Omron CX-Programmer project NewProject (CX-Programmer 9.73)

# PLC NewPLC1: CJ1M CPU11

## Global symbols (name address type ; comment)
At_exit_forward 0.10 BOOL
At_exit_left 0.09 BOOL
At_exit_right 0.11 BOOL
At_forward_entry 0.07 BOOL
At_left_entry 0.06 BOOL
At_right_entry 0.08 BOOL
At_scale 0.04 BOOL
At_scale_entry 0.03 BOOL
At_scale_exit 0.05 BOOL
W200 CHANNEL  ; weight_help
Emergency 0.02 BOOL
Entry_conveyor W1.00 BOOL
Entry_conveyor_act 1.00 BOOL  ; Entry_conveyor
Forward_conveyor W1.03 BOOL
Forward_conveyor_act 1.03 BOOL
Forward_counter W301 INT
Forward_screen 2 CHANNEL
Left_conveyor W1.02 BOOL
Left_conveyor_act 1.02 BOOL
Left_counter W300 INT
Left_screen 1 CHANNEL
Load_scale W1.01 BOOL
Load_scale_act 1.01 BOOL
Mid W100 INT
Mid_flag W1.05 BOOL
On_forward_conveyor W304 INT
On_forward_conveyor_minus W1.08 BOOL
On_left_conveyor W303 INT
On_left_conveyor_minus W1.07 BOOL
On_load_scale W306 INT
On_load_scale_minus W1.06 BOOL
On_right_conveyor W305 INT
On_right_conveyor_minus W1.09 BOOL
Program_entry W0.01 BOOL
Right_conveyor W1.04 BOOL
Right_conveyor_act 1.04 BOOL
Right_counter W302 INT
Right_screen 3 CHANNEL
Start 0.00 BOOL  ; start
Stop 0.01 BOOL
Weight W0 INT  ; weight
Weight_screen 4 CHANNEL

## Program weight_sorter_program (cyclic task 1)
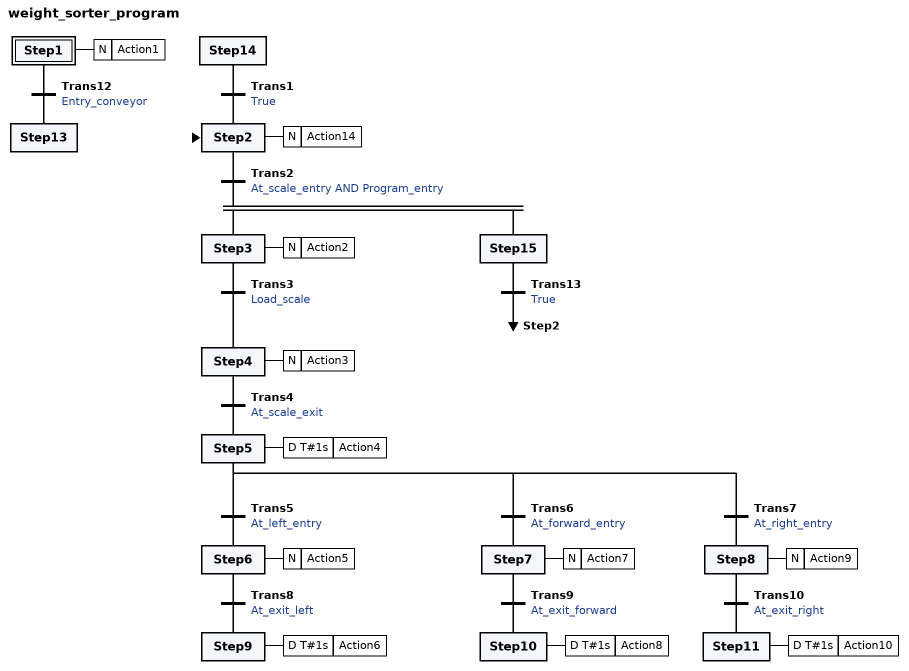
INITIAL_STEP Step1 :
Action1(N) ;
END_STEP
TRANSITION Trans1 FROM Step14 TO Step2
 := True;
END_TRANSITION
STEP Step2 :
Action14(N) ;
END_STEP
TRANSITION Trans2 FROM Step2 TO (Step3,Step15)
 := At_scale_entry AND Program_entry;
END_TRANSITION
STEP Step3 :
Action2(N) ;
END_STEP
TRANSITION Trans3 FROM Step3 TO Step4
 := Load_scale;
END_TRANSITION
STEP Step4 :
Action3(N) ;
END_STEP
TRANSITION Trans4 FROM Step4 TO Step5
 := At_scale_exit;
END_TRANSITION
STEP Step5 :
Action4(D,T#1s) ;
END_STEP
TRANSITION Trans5 (PRIORITY := 1) FROM Step5 TO Step6
 := At_left_entry;
END_TRANSITION
TRANSITION Trans6 (PRIORITY := 2) FROM Step5 TO Step7
 := At_forward_entry;
END_TRANSITION
TRANSITION Trans7 (PRIORITY := 3) FROM Step5 TO Step8
 := At_right_entry;
END_TRANSITION
STEP Step6 :
Action5(N) ;
END_STEP
TRANSITION Trans8 FROM Step6 TO Step9
 := At_exit_left;
END_TRANSITION
STEP Step7 :
Action7(N) ;
END_STEP
TRANSITION Trans9 FROM Step7 TO Step10
 := At_exit_forward;
END_TRANSITION
STEP Step8 :
Action9(N) ;
END_STEP
TRANSITION Trans10 FROM Step8 TO Step11
 := At_exit_right;
END_TRANSITION
STEP Step9 :
Action6(D,T#1s) ;
END_STEP
STEP Step10 :
Action8(D,T#1s) ;
END_STEP
STEP Step11 :
Action10(D,T#1s) ;
END_STEP
TRANSITION Trans12 FROM Step1 TO Step13
 := Entry_conveyor;
END_TRANSITION
STEP Step14 :
END_STEP
STEP Step15 :
END_STEP
TRANSITION Trans13 FROM Step15 TO Step2
 := True;
END_TRANSITION
STEP Step13 :
END_STEP

### Action Action1

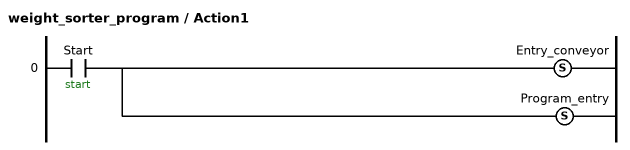
; rung 0
LD Start  ; start
SET Entry_conveyor
SET Program_entry

### Action Action2

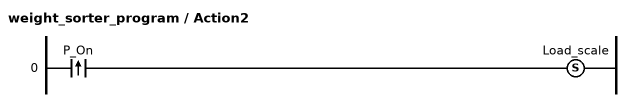
; rung 0
@LD P_On
SET Load_scale

### Action Action3

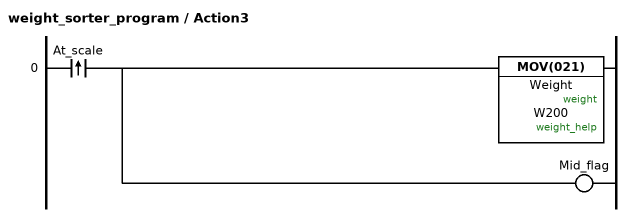
; rung 0
@LD At_scale
MOV(021) Weight W200  ; weight, weight_help
OUT Mid_flag

### Action Action4

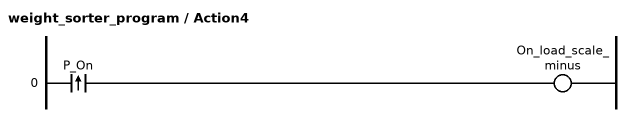
; rung 0
@LD P_On
OUT On_load_scale_minus

### Action Action5

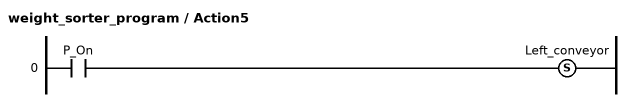
; rung 0
LD P_On
SET Left_conveyor

### Action Action6

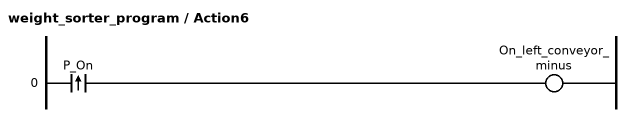
; rung 0
@LD P_On
OUT On_left_conveyor_minus

### Action Action7

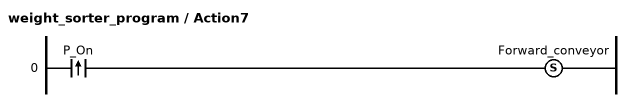
; rung 0
@LD P_On
SET Forward_conveyor

### Action Action8

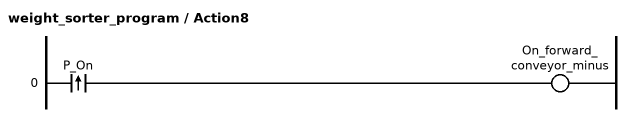
; rung 0
@LD P_On
OUT On_forward_conveyor_minus

### Action Action9

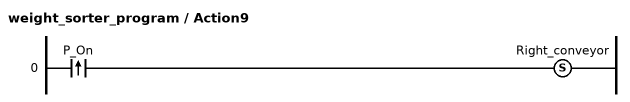
; rung 0
@LD P_On
SET Right_conveyor

### Action Action10

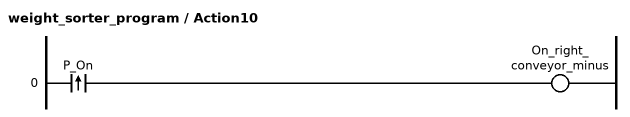
; rung 0
@LD P_On
OUT On_right_conveyor_minus

### Action Action11

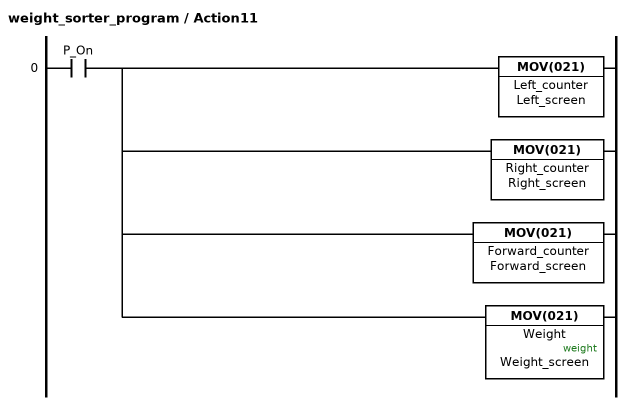
; rung 0
LD P_On
MOV(021) Left_counter Left_screen
MOV(021) Right_counter Right_screen
MOV(021) Forward_counter Forward_screen
MOV(021) Weight Weight_screen  ; weight

### Action Action12

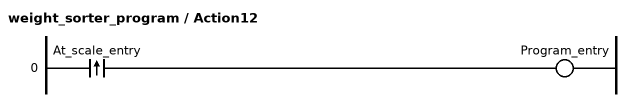
; rung 0
@LD At_scale_entry
OUT Program_entry

### Action Action13

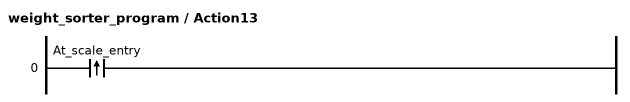
; rung 0
@LD At_scale_entry

### Action Action14

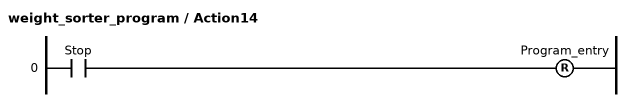
; rung 0
LD Stop
RSET Program_entry

### Action Action15

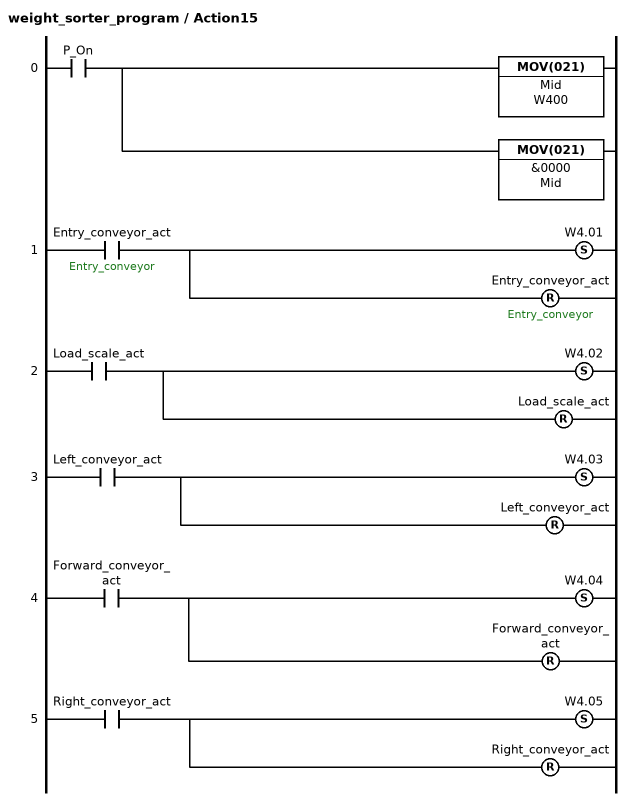
; rung 0
LD P_On
MOV(021) Mid W400
MOV(021) &0000 Mid
; rung 1
LD Entry_conveyor_act  ; Entry_conveyor
SET W4.01
RSET Entry_conveyor_act  ; Entry_conveyor
; rung 2
LD Load_scale_act
SET W4.02
RSET Load_scale_act
; rung 3
LD Left_conveyor_act
SET W4.03
RSET Left_conveyor_act
; rung 4
LD Forward_conveyor_act
SET W4.04
RSET Forward_conveyor_act
; rung 5
LD Right_conveyor_act
SET W4.05
RSET Right_conveyor_act

### Action Action16

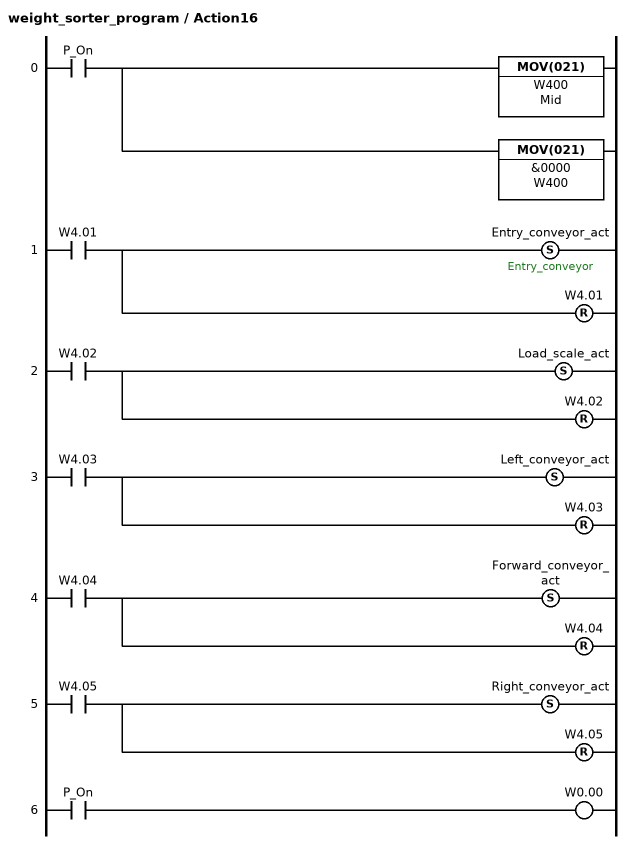
; rung 0
LD P_On
MOV(021) W400 Mid
MOV(021) &0000 W400
; rung 1
LD W4.01
SET Entry_conveyor_act  ; Entry_conveyor
RSET W4.01
; rung 2
LD W4.02
SET Load_scale_act
RSET W4.02
; rung 3
LD W4.03
SET Left_conveyor_act
RSET W4.03
; rung 4
LD W4.04
SET Forward_conveyor_act
RSET W4.04
; rung 5
LD W4.05
SET Right_conveyor_act
RSET W4.05
; rung 6
LD P_On
OUT W0.00

## Program NewProgram1 (cyclic task 0)

### Section Section1

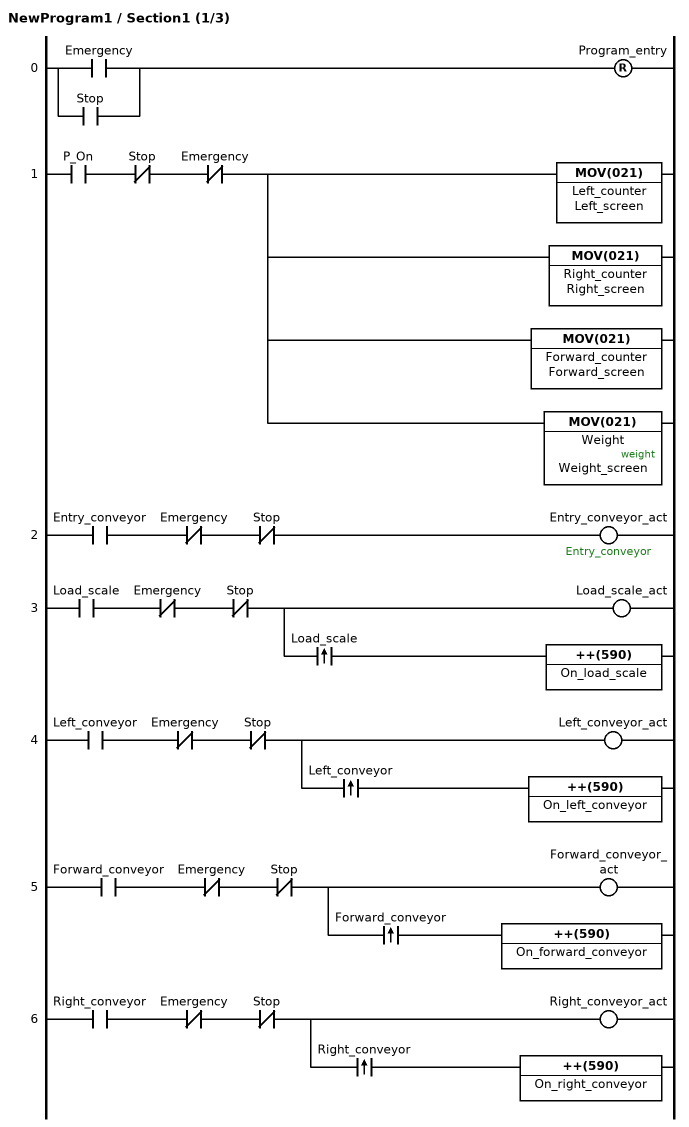
; rung 0
LD Emergency
OR Stop
RSET Program_entry
; rung 1
LD P_On
ANDNOT Stop
ANDNOT Emergency
MOV(021) Left_counter Left_screen
MOV(021) Right_counter Right_screen
MOV(021) Forward_counter Forward_screen
MOV(021) Weight Weight_screen  ; weight
; rung 2
LD Entry_conveyor
ANDNOT Emergency
ANDNOT Stop
OUT Entry_conveyor_act  ; Entry_conveyor
; rung 3
LD Load_scale
ANDNOT Emergency
ANDNOT Stop
OUT Load_scale_act
@AND Load_scale
++(590) On_load_scale
; rung 4
LD Left_conveyor
ANDNOT Emergency
ANDNOT Stop
OUT Left_conveyor_act
@AND Left_conveyor
++(590) On_left_conveyor
; rung 5
LD Forward_conveyor
ANDNOT Emergency
ANDNOT Stop
OUT Forward_conveyor_act
@AND Forward_conveyor
++(590) On_forward_conveyor
; rung 6
LD Right_conveyor
ANDNOT Emergency
ANDNOT Stop
OUT Right_conveyor_act
@AND Right_conveyor
++(590) On_right_conveyor

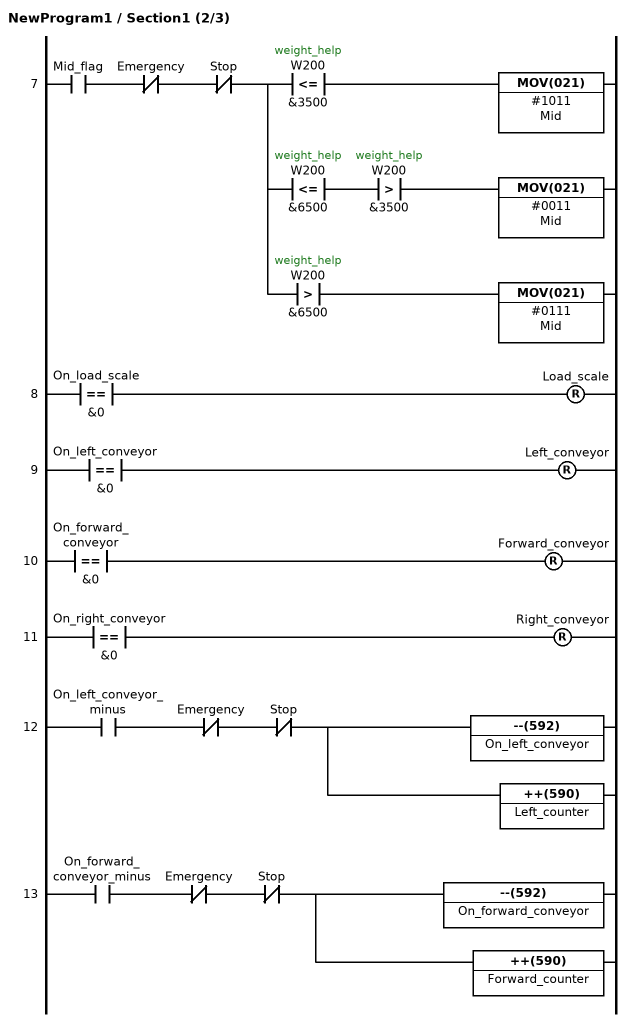
; rung 7
LD Mid_flag
ANDNOT Emergency
ANDNOT Stop
OUT TR0
AND<=(315) W200 &3500  ; weight_help
MOV(021) #1011 Mid
LD TR0
AND<=(315) W200 &6500  ; weight_help
AND>(320) W200 &3500  ; weight_help
MOV(021) #0011 Mid
LD TR0
AND>(320) W200 &6500  ; weight_help
MOV(021) #0111 Mid
; rung 8
LD=(300) On_load_scale &0
RSET Load_scale
; rung 9
LD=(300) On_left_conveyor &0
RSET Left_conveyor
; rung 10
LD=(300) On_forward_conveyor &0
RSET Forward_conveyor
; rung 11
LD=(300) On_right_conveyor &0
RSET Right_conveyor
; rung 12
LD On_left_conveyor_minus
ANDNOT Emergency
ANDNOT Stop
--(592) On_left_conveyor
++(590) Left_counter
; rung 13
LD On_forward_conveyor_minus
ANDNOT Emergency
ANDNOT Stop
--(592) On_forward_conveyor
++(590) Forward_counter

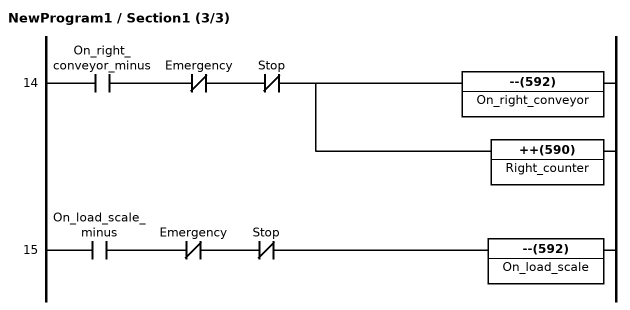
; rung 14
LD On_right_conveyor_minus
ANDNOT Emergency
ANDNOT Stop
--(592) On_right_conveyor
++(590) Right_counter
; rung 15
LD On_load_scale_minus
ANDNOT Emergency
ANDNOT Stop
--(592) On_load_scale

### Section END
; rung 0
END(001)